TYPE ST_CamTable :
STRUCT
	TableData 		: ARRAY [0..360,0..1] OF LREAL;
	Id				: UDINT;
	Rows			: UDINT;
	Periodic		: BOOL;
	Generate		: BOOL;
	//StartMode		: MC_StartMode;
END_STRUCT
END_TYPE

(* stored: Version 1.1.0.1, ProductVersion 3.1.4024.3
   DUT ST_CamTable: Id {a0f802b0-37b5-4fdb-9c7c-6c77f0976289} *)
